{attribute 'obsolete' := 'Use E_EpicsHomeCmd'}
TYPE ENUM_EpicsHomeCmd : E_EpicsHomeCmd; END_TYPE

(* stored: Version 1.1.0.1
   DUT ENUM_EpicsHomeCmd: Id {d3cf1823-84b7-4d07-a230-30e3b5f14b37} *)
